(* CODESYS project basevista.library
   Company: Vistaprint
   Title: Base_PLC
   Description: 0.3.4.8 - Bug fix alarm entry,reset and clear
      0.3.4.7 - Increased the maxchildnumber to 40
      0.3.4.6 - Increased the maxchildnumber to 40
      0.3.4.5 - BugFix in alarm manager
      0.3.4.2 - Changed the Pramas Text in FB_CtrlBase
      0.3.4.1 - State single answer. Reset pending alarm class to NONE.
      0.3.4.0 - New CheckAllChildState also true feedback if check state of child OFF or EOFF and child in ERROR;
      - Bug fix Always Single-answer and startup with wait on PON
      - FB_Alm_Man: New Property IsInitDone		feedback at least one valid time stamp read out 
      0.3.3.7 - CheckParentAlmClass OFF and STOP added -> reaction of Controller
      0.3.3.6 - FB_Alm_Man Property CntPerClass added, alarm classes EOFF, OFF and STOP from parent to child, in EOFFBusy and OFF busy command in cyclic action (not entry action)
      
      0.3.3.4 - Added IO support for USINT datatype
      
      0.3.3.3 - Bug fixed in getInBolDebounced(FUN)
      
      0.3.3.2 - New function setAllCtrlAlarmFB -> all controller init pointer of alarmhandler; 
      - Rename GetInUint ->getInUint; 
      - New function ScaleINT (scale integer variable p.e. analog increment to 0.1mm)
      
      0.3.3.1  Added getInBolDebounced(FUN) and T_Ctrl_IoBoolDebounced(STRUCT) for debouncing inputs
      0.3.3.0 - Added pfbAlarmCtrl and the "zugehörige" property to allow clean alarm calls also from controllers in libraries.
      0.3.2.0 - Del getCtrlCIF,iniCtrlArray; Set cmds to child EOFF,OFF,PON; EOFF State; Check child ALM EOFF     
      0.3.1.3 - Bugfix
      0.3.1.2 - Added iniAllCtrlArrays - this is iniCtrlArray + the cif array
      0.3.1 - Added the automatic EOff propagation.
      0.3.0 - Added the substate to T_CTRL_CLASS_STATEMACHINE
      Automatic Substate handling.
      0.2.3 - Added support for sub usec cycletimes
      0.2.2 - Added the UInt for IO. T_CTRL_IOUint, setInUint(), setOutUint()
      0.2.1 - Added the property CtrlCIf to FB_CtrlBase
   Version: 0.3.4.8

Project tree, tasks and I/O mapping:
  libraries: Tc2_Standard, 3.3.0.0 (Beckhoff Automation GmbH); Tc2_System, 3.3.5.0 (Beckhoff Automation GmbH); Tc2_Utilities, 3.3.7.0 (Beckhoff Automation GmbH); Tc3_Interfaces, 3.3.0.0 (Beckhoff Automation GmbH); Tc3_MemMan, 3.3.1.0 (Beckhoff Automation GmbH); Tc3_Module, 3.3.5.0 (Beckhoff Automation GmbH)
  POUs/
    Alarm/
      data type E_AlmClass
      data type E_AlmCmd
      data type E_AlmState
      function block FB_Alm_Man [ST]: aCntPerClass, clearAlarm, IsInitDone, setAlarm
      data type T_AlmElement
      data type T_Ctrl_Alm
    BaseCtrl/
      global variables Base_CmdState
      global variables Base_Const
      data type E_Mode
      function block FB_CtrlBase [ST]: AddChild, AlarmCtrl, Always, CheckAllChildAlmClass, CheckAllChildState, CheckChildAlmClass, CheckCmdValid, CheckParentAlmClass, CtrlCIf, CtrlFB, CtrlInit, CycleEndDuty, CycleStartDuty, EOFF_EntryAction, FB_init, getCmdState, iniAllCtrlArrays, IoInBridge, IoOutBridge, SetAllChildAlmClass, SetAllChildCmd, sta_EOFF, sta_EOFFBusy, sta_ERROR, sta_ERRORQuit, sta_OFF, sta_OFFBusy, sta_PON, sta_PONBusy, sta_SINGLE_ANSWER, StateMachine
      interface I_CtrlBase: CtrlCIf, CtrlFB
      data type T_Ctrl_CIf
      data type T_Ctrl_Class
      data type T_Ctrl_Class_Alm
      data type T_Ctrl_Class_StateMachine
      data type T_Ctrl_CmdListElement
      data type T_Ctrl_Info
      data type T_Ctrl_IoBool
      data type T_Ctrl_IoBoolDebounced
      data type T_Ctrl_IoInt
      data type T_Ctrl_IoUint
      data type T_Ctrl_IoUsint
      data type T_Ctrl_Job
      data type T_Ctrl_SwCfg
      data type T_fbInfo
    Utility/
      DLL (Double Linked List)/
        function block FB_DLL [ST]: addElement, deleteAll, deleteElement, FB_init, firstElement, numberOfElements, searchElement
        data type T_Element
      function getInBol [ST]
      function getInBolDebounced [ST]
      function getInInt [ST]
      function getInUint [ST]
      function getInUsint [ST]
      function getStrInstanceName [ST]
      function ScaleINT [ST]
      function setAllCtrlAlarmFB [ST]
      function setOutBol [ST]
      function setOutInt [ST]
      function setOutUint [ST]
      function setOutUsint [ST]
  Version/
    global variables Global_Version
*)

// POUs/Alarm/E_AlmClass
TYPE E_AlmClass :
(
	///no alarm active
	NONE := 0,
	///info
	INFO,
	///warning
	WARNING,
	///tact stop
	TSTOP,
	///stop
	STOP,
	///off
	OFF,
	///Emergency off
	EOFF,
	Max_E_AlmClass
) INT;
END_TYPE

// POUs/Alarm/E_AlmCmd
TYPE E_AlmCmd :
(
	DONE := -1,
	INITIALIZED := 0,
	RESET_ALL := 2,
	RESET_RST := 4,
	RESET_CLR := 6,
	Max_E_AlmCmd
);
END_TYPE

// POUs/Alarm/E_AlmState
TYPE E_AlmState :
(
	///no alarm active
	NONE := 0,
	///alarm clear entry -> set bit1
	CLR := 1,
	///entry resettable alarm ->  set bit2
	RST := 2,
	///entry non resettable alarm ->  set bit2 + bit3
	SET := 3,
	Max_E_AlmState
);
END_TYPE

// POUs/Alarm/T_AlmElement
TYPE T_AlmElement :
STRUCT
	///unique alarm number := 100000*udiMachineNr + intCtrlId*100 + udiAlarmNr
	udiNr: UDINT;
	///additional information - better string???
	dinInfo: DINT;
	///corresponding alarm class
	eClass: E_AlmClass;
	///clear, resetable
	intState: E_AlmState;
	///entry time
	strDTEntry: STRING;
	///from machine (standard = 1)
	udiMachineNr: UDINT;
	///from controller
	intCtrlId: INT;
	///local alarm number
	udiAlarmNr: UDINT;
	// for debugging string alarm controller-alarm
	strText: STRING;
END_STRUCT
END_TYPE

// POUs/Alarm/T_Ctrl_Alm
TYPE T_Ctrl_Alm :
STRUCT
	///alarm flag array
	bol: BOOL;
	eAlmClass: E_AlmClass;
	strText: STRING;
END_STRUCT
END_TYPE

// POUs/BaseCtrl/E_Mode
{attribute 'qualified_only' := ''}
TYPE E_Mode :
(
	INITIALIZED := 0,
	AUTO := 10,
	SEMI := 11,
	MANU := 12
) INT;
END_TYPE

// POUs/BaseCtrl/T_Ctrl_CIf
TYPE T_Ctrl_CIf :
STRUCT
	Job: T_Ctrl_Job;
	Info: T_Ctrl_Info;
	SwCfg: T_Ctrl_SwCfg;
END_STRUCT
END_TYPE

// POUs/BaseCtrl/T_Ctrl_Class
TYPE T_Ctrl_Class :
STRUCT
	///local test flag to supress cyclic run (for debugging after init)
	bolActivate					: BOOL;
	intCmd						: INT;
	intCmdLast					: INT;
	eModeHistory				: E_Mode;
	///local flag mode change detected
	bolChangeBackToAUTO			: BOOL;
	StateMachine				: T_Ctrl_Class_StateMachine;
	SubStateMachine				: T_Ctrl_Class_StateMachine;
	Alarm						: T_Ctrl_Class_Alm;
	FUBInfo						: T_fbInfo;
END_STRUCT
END_TYPE

// POUs/BaseCtrl/T_Ctrl_Class_Alm
TYPE T_Ctrl_Class_Alm :
STRUCT
	bolResetOk: BOOL;
	///flag positive check me alarm from child
	bolfp: BOOL;
	///local activ alarm class of parent ctrl
	eParent_ActivAlmClass: E_AlmClass;
	///highest local activ alarm class
	eActivAlmClass: E_AlmClass;
END_STRUCT
END_TYPE

// POUs/BaseCtrl/T_Ctrl_Class_StateMachine
TYPE T_Ctrl_Class_StateMachine :
STRUCT
	///actual state
	intState: INT;
	///state of last cycle
	intStateLastCycle: INT;
	///save history backup p.e. in ERROR state
	intStateHistory: INT;
	///set state for next cycle
	intStateNext: INT;
	///[ms] to simulate state in SINGLE_ANSWER
	udiStateSimSetTime_ms: UDINT := 1000;
	///[ms] time in one state
	udiTimeInState_ms: UDINT;
	///[ms] time in one state
	relTimeInState_ms: REAL;
	///[us] time in one state
	udiTimeInState_us: UDINT;
END_STRUCT
END_TYPE

// POUs/BaseCtrl/T_Ctrl_CmdListElement
TYPE T_Ctrl_CmdListElement :
STRUCT
	///command implemented in controller
	intCmd: INT;
	///command is available info for UI
	bolAvailable: BOOL;
	/// Name of command. Important for UI.
	strName: STRING(80);
END_STRUCT
END_TYPE

// POUs/BaseCtrl/T_Ctrl_Info
TYPE T_Ctrl_Info :
STRUCT
	///name of controller instance
	strName				: STRING(80);
	///class of controller
	strType				: STRING(80);
	///unique controller instance identification number
	intCtrlId			: INT;
	///unique identification number of parent controller instance
	intParentCtrlId		: INT;
	///all inputs valid -> init done
	bolInitDone			: BOOL;
	///Childs
	p_afbChild			: ARRAY[0..Base_Const.cMaxNrOfChilds] OF POINTER TO FB_CtrlBase;
	///common interface array of childs
	p_aCIf				: ARRAY[0..Base_Const.cMaxNrOfChilds] OF POINTER TO T_Ctrl_CIf;
	/// Child Count
	uinChildNbr			: UINT;
END_STRUCT
END_TYPE

// POUs/BaseCtrl/T_Ctrl_IoBool
TYPE T_Ctrl_IoBool :
STRUCT
	///mapped io variable to hardware
	map: BOOL;
	///shows the state of (input: mapped, output: set by programm respectiv at the moment one cycle later evtl. from the forcing if forcing active) -> necessary for what?
	state: BOOL;
	///variabel to/ from program
	intern: BOOL;
	///variabel set from UI
	force: BOOL;
	///enable force of single io-datapoint
	EnForce: BOOL;
END_STRUCT
END_TYPE

// POUs/BaseCtrl/T_Ctrl_IoBoolDebounced
TYPE T_Ctrl_IoBoolDebounced :
STRUCT
	///mapped io variable to hardware
	map: BOOL;
	///shows the state of (input: mapped, output: set by programm respectiv at the moment one cycle later evtl. from the forcing if forcing active) -> necessary for what?
	state: BOOL;
	///variabel to/ from program
	intern: BOOL;
	///variabel set from UI
	force: BOOL;
	///enable force of single io-datapoint
	EnForce: BOOL;
	// time since last input change
	udinDebouncedTimeCounter_ms: UDINT;
END_STRUCT
END_TYPE

// POUs/BaseCtrl/T_Ctrl_IoInt
TYPE T_Ctrl_IoInt :
STRUCT
	///mapped io variable to hardware
	map: INT;
	///shows the state of (input: mapped, output: set by programm respectiv at the moment one cycle later evtl. from the forcing if forcing active) -> necessary for what?
	state: INT;
	///variabel to/ from program
	intern: INT;
	///variabel set from UI
	force: INT;
	///enable force of single io-datapoint
	EnForce: BOOL;
END_STRUCT
END_TYPE

// POUs/BaseCtrl/T_Ctrl_IoUint
TYPE T_Ctrl_IoUint :
STRUCT
	///mapped io variable to hardware
	map: UINT;
	///shows the state of (input: mapped, output: set by programm respectiv at the moment one cycle later evtl. from the forcing if forcing active) -> necessary for what?
	state: UINT;
	///variabel to/ from program
	intern: UINT;
	///variabel set from UI
	force: UINT;
	///enable force of single io-datapoint
	EnForce: BOOL;
END_STRUCT
END_TYPE

// POUs/BaseCtrl/T_Ctrl_IoUsint
TYPE T_Ctrl_IoUsint :
STRUCT
	///mapped io variable to hardware
	map: USINT;
	///shows the state of (input: mapped, output: set by programm respectiv at the moment one cycle later evtl. from the forcing if forcing active) -> necessary for what?
	state: USINT;
	///variabel to/ from program
	intern: USINT;
	///variabel set from UI
	force: USINT;
	///enable force of single io-datapoint
	EnForce: BOOL;
END_STRUCT
END_TYPE

// POUs/BaseCtrl/T_Ctrl_Job
TYPE T_Ctrl_Job :
STRUCT
	///mode if mode = AUTO -> ACmd will be used, otherwise the MCmd channel is open
	eMode: E_Mode;
	///automatic command from parent ctrl
	intACmd: INT;
	///manual command from UI p.e.
	intMCmd: INT;
	///active cmd
	strCmd: STRING;
	///active state
	intState: INT;
	strState: STRING;
	///if used - show substates for debugging
	strSubState: STRING;
	///event channel to signal special events to parent parallel to status
	intEvt: INT;
	///reset all alarms
	bolAlmReset: BOOL;
	///activate io-forcing
	bolIoForce: BOOL;
	///overwrite suspend all interlocks (for debugging/testing)
	bolIlkOverwrite: BOOL;
	///activ alarm class of parent ctrl
	eParent_ActivAlmClass: E_AlmClass;
	///activ alarm class of me ctrl
	eMe_ActivAlmClass: E_AlmClass;
	///list of all implemented commands
	aCmdList: ARRAY[0..cMaxCmdPerCtrl] OF T_Ctrl_CmdListElement;
END_STRUCT
END_TYPE

// POUs/BaseCtrl/T_Ctrl_SwCfg
TYPE T_Ctrl_SwCfg :
	STRUCT
		///hardware/controller exists
		bolExist: BOOL;
		///enable statemachine
		bolEnable: BOOL;
		///set controller in simulation(statemachine active, io local simulated)
		bolSimulation: BOOL;
	END_STRUCT
END_TYPE

// POUs/BaseCtrl/T_fbInfo
TYPE T_fbInfo :
STRUCT
	bolCycleTimeBelowMS			: BOOL;
	udiSample_ms				: UDINT;
	udiSample_us				: UDINT;
END_STRUCT
END_TYPE

// POUs/Utility/DLL (Double Linked List)/T_Element
{attribute 'enable_dynamic_creation' := ''}
TYPE T_Element :
STRUCT
	pPrevElement: POINTER TO T_Element;
	pData: POINTER TO BYTE;
	uliKey: ULINT;
	pNextElement: POINTER TO T_Element;
END_STRUCT
END_TYPE

// POUs/BaseCtrl/Base_CmdState
VAR_GLOBAL CONSTANT
	///ctrl commands definitions
	///general commands 2-200 - every command has to be a even number
	cCMD_DONE: INT := -1;
	cCMD_INITIALIZED: INT := 0;
	cCMD_PON: INT := 2;
	cCMD_EOFF: INT := 4;
	cCMD_OFF: INT := 6;
	cCMD_INIT: INT := 8;
	cCMD_RUN: INT := 10;
	cCMD_STOP: INT := 12;
	cCMD_TSTOP: INT := 14;
	///ctrl states definitions
	cSTA_DONE: INT := cCMD_DONE;
	cSTA_INITIALIZED: INT := cCMD_INITIALIZED;
	cSTA_PONBusy: INT := 1;
	cSTA_PON: INT := cCMD_PON;
	cSTA_EOFFBusy: INT := 3;
	cSTA_EOFF: INT := cCMD_EOFF;
	cSTA_OFFBusy: INT := 5;
	cSTA_OFF: INT := cCMD_OFF;
	cSTA_INITBusy: INT := 7;
	cSTA_INIT: INT := cCMD_INIT;
	cSTA_RUNBusy: INT := 9;
	cSTA_RUN: INT := cCMD_RUN;
	cSTA_STOPBusy: INT := 11;
	cSTA_STOP: INT := cCMD_STOP;
	cSTA_TSTOPBusy: INT := 13;
	cSTA_TSTOP: INT := cCMD_TSTOP;
	///special states without corresponding cmd
	cSTA_ERROR: INT := 150;
	cSTA_ERRORQuit: INT := 151;
	cSTA_SINGLE_ANSWER: INT := 152;
END_VAR

// POUs/BaseCtrl/Base_Const
VAR_GLOBAL CONSTANT
	///number of child access possible in one controller class
	cMaxNrOfChilds: UINT := 25;
	///maximal number of commands implemented in one controller class
	cMaxCmdPerCtrl: UINT := 15;
	///maximal number of commands implemented in one controller class
	cMaxBaseCmdState: UINT := 200;
END_VAR

// Version/Global_Version
// This function has been automatically generated from the project information.
VAR_GLOBAL CONSTANT
	{attribute 'const_non_replaced'}
	stLibVersion_Base_PLC : ST_LibVersion := (iMajor := 0, iMinor := 3, iBuild := 4, iRevision := 8, sVersion := '0.3.4.8');
END_VAR

// POUs/Alarm/FB_Alm_Man
FUNCTION_BLOCK FB_Alm_Man
VAR_INPUT
	;
END_VAR
VAR_IN_OUT
	bolCtrlRst: BOOL; // reset all controller
END_VAR

VAR CONSTANT
	/// config alarm handler number of elements of queue
	c_uinMaxAlmElements: UINT := 99;
	/// 0: with history on PLC, auto clr alarms from array if alarm state clear is set
	c_uinModeAlarm: UINT := 1;
	/// machine number 1, at the moment every time set to 1
	c_udiMachineNr: UDINT := 1;
	/// commands from the UI
	cCMD_RESET_ALL: INT := 2;
	/// reset state=RST, reset state CLR
	cCMD_RESET_RST: INT := 4;
	/// reset state CLR -> c_uinModeAlarm = 1, automatic reset will be done on PLC
	cCMD_RESET_CLR: INT := 6;
END_VAR
VAR
	///------------------------------------------------------------
	/// UI interface
	/// alarmarray PLC -> UI
	aAlm: ARRAY[0..c_uinMaxAlmElements] OF T_AlmElement;
	/// command interface for UI -> PLC
	intAlmCmd: INT;
	///------------------------------------------------------------
	/// real local variables
	fbGetLocalTime: NT_GetTime;
	strActTime: STRING;
	jj: UINT;
	EmptyAlmElement: T_AlmElement;
	intState: INT;
	intTestCtrl: INT := 12;
	intTestState: INT;
	udiTestAlarmNr: UDINT;
	dinTestInfo: DINT;
	aCtrlAlm: ARRAY[1..6] OF T_Ctrl_Alm;
	eActiveAlmClass: E_AlmClass;

	aCntActiveAlmPerClass: ARRAY[0..(E_AlmClass.Max_E_AlmClass-1)] OF UINT; // count off all active alarms per class, idx=0 all active alarms
	bolTimeReadDone : BOOL;
	bolTimeStampValid : BOOL;
END_VAR

(*__________________________________________________________________________________________________
¦	
¦	Vistaprint Schweiz GmbH
¦	CH - 8401 Winterthur
¦
¦	www.vistaprint.ch - info@vistaprint.ch
¦___________________________________________________________________________________________________

Function desription:
The alarm manager sets and clears alarms from the internal array. In the internal array all active 
alarms of a machine are listed. The list has no order. A new entry will be inserted at the next 
free place.

For the easy usage for UI the function block is to be define as global. And then the cmd for reset should be 
set when the button is pressed -> intAlmCmd = cCMD_RESET_ALL
All active alarms are shown in the aAlm array.

History:
Version		Date			Author		Comment
---------------------------------------------------------------------------------------------------
0.00.1		29.04.2013		AVME/KVO	Start history
0.00.2		06.01.2014		AVME/PRE	Implement the counted active messages array
0.00.3		17.02.2014		AVME/KVO	New Property IsInitDone 
										feedback at least one valid time stamp read out 
										-> check at startup before cyclic call of FB's to avoid alarms without valid timestamp
0.00.4		16.05.2014		AVME/DSC	-> Inserted new "setAlarm" Method from Patrik C. (code review)									
										-> BugFix, build sum of all active alarms
___________________________________________________________________________________________________*)

// read out actual TIME
fbGetLocalTime.NETID := '';
fbGetLocalTime.START := NOT bolTimeReadDone;
fbGetLocalTime.TMOUT := T#5S;
fbGetLocalTime();

IF (fbGetLocalTime.START=TRUE) THEN
	IF  ((fbGetLocalTime.Busy=FALSE) AND (fbGetLocalTime.ERR=FALSE)) THEN
		bolTimeReadDone := TRUE;
		strActTime := TC2_UTILITIES.SYSTEMTIME_TO_STRING(fbGetLocalTime.TIMESTR); // YYYY-MM-DD-hh:mm:ss.xxx
		bolTimeStampValid := TRUE; // -> entry alarms with valid time stamp
	END_IF
ELSE
	bolTimeReadDone := FALSE;
END_IF


// interface for UI access
CASE intState OF
	
	0: // reset cmd
		intAlmCmd := cCMD_DONE; // Ready for new cmd
		intState := intState + 1;
		
	1: // wait for cmd
		IF (intAlmCmd=cCMD_RESET_ALL) OR (intAlmCmd=cCMD_RESET_CLR) OR  (intAlmCmd=cCMD_RESET_RST) THEN
			intState := intState + 1;
		END_IF
		
	2: // reset alarms
		// reset state=RST, reset state CLR
		THIS^.clearAlarm(((intAlmCmd=cCMD_RESET_ALL) OR (intAlmCmd=cCMD_RESET_RST)), TRUE);
		intState := intState + 1;
		
	3: // reset state machines
		bolCtrlRst := TRUE;
		intState := 0; // done

END_CASE

// build sum of all active alarms
aCntActiveAlmPerClass[0] := 0;
FOR jj:= 1 TO INT_TO_UINT(E_AlmClass.Max_E_AlmClass-1) BY 1 DO
	aCntActiveAlmPerClass[0] := aCntActiveAlmPerClass[0] + aCntActiveAlmPerClass[jj];
END_FOR

//**********************************************************************************************
// Test manual set/reset/clear alarm
//**********************************************************************************************
CASE intTestState OF
	
	0: // wait
		
	1: //CLR
		THIS^.setAlarm(intTestCtrl,udiTestAlarmNr,dinTestInfo,ADR(aCtrlAlm),E_AlmState.CLR,eActiveAlmClass);
		intTestState := 0;
		
	2: // RST
		THIS^.setAlarm(intTestCtrl,udiTestAlarmNr,dinTestInfo,ADR(aCtrlAlm),E_AlmState.RST,eActiveAlmClass);
		intTestState := 0;
		
	3: // SET
		THIS^.setAlarm(intTestCtrl,udiTestAlarmNr,dinTestInfo,ADR(aCtrlAlm),E_AlmState.SET,eActiveAlmClass);
		intTestState := 0;

END_CASE

PROPERTY PUBLIC aCntPerClass : ARRAY[0..(E_AlmClass.Max_E_AlmClass-1)] OF UINT
GET
aCntPerClass := aCntActiveAlmPerClass;
END_GET
END_PROPERTY

METHOD clearAlarm : BOOL
VAR_INPUT
	///-> clear all entries with state RST
	bolClear_RST: BOOL;
	///-> clear all entries with state CLR
	bolClear_CLR: BOOL;
END_VAR
VAR
	ii: UINT;
END_VAR
FOR ii:= 0 TO INT_TO_UINT(E_AlmClass.Max_E_AlmClass-1) BY 1 DO
	aCntActiveAlmPerClass[ii] := 0; // reset alarm counter
END_FOR

FOR ii:= 0 TO c_uinMaxAlmElements BY 1 DO
	
	IF (aAlm[ii].udiNr>0) THEN 
		
		IF (((aAlm[ii].intState=E_AlmState.RST) AND (bolClear_RST)) OR
			((aAlm[ii].intState=E_AlmState.CLR) AND (bolClear_CLR)))THEN
			
			aAlm[ii] := EmptyAlmElement; // clear entry
		ELSE
			//count alarms per class
			aCntActiveAlmPerClass[aAlm[ii].eClass] := aCntActiveAlmPerClass[aAlm[ii].eClass] + 1; 
		END_IF
		
	END_IF
END_FOR
END_METHOD

PROPERTY IsInitDone : BOOL
GET
// feedback at least one valid time stamp read out 
//-> check at startup before cyclic call of FB's to avoid alarms without valid timestamp
IsInitDone := bolTimeStampValid;
END_GET
END_PROPERTY

METHOD setAlarm : E_AlmClass
VAR_INPUT
	///from controller 
	intCtrlId: INT;
	///local alarm number
	udiAlarmNr: UDINT;
	///additional information - string???
	dinInfo: DINT;
	///corresponding alarm class
	p_Ctrl_Alm: POINTER TO T_Ctrl_Alm;
	///clear, resetable
	intState: E_AlmState;
END_VAR
VAR_IN_OUT
	eMe_ActivAlmClass: E_AlmClass;
END_VAR
VAR
	InAlmElement: T_AlmElement;
	ii: UINT;
	e_LocAlmClass: E_AlmClass;
END_VAR
// chack if pointer valid
IF (p_Ctrl_Alm <> Tc3_MemMan.NULL) AND (udiAlarmNr>0) THEN 
	e_LocAlmClass := p_Ctrl_Alm[udiAlarmNr-1].eAlmClass;
ELSE
	// novalid pointer reached!!
   	e_LocAlmClass := E_AlmClass.EOFF; 
END_IF
 
// Copy alarm input data to local alm struct
InAlmElement.udiMachineNr := c_udiMachineNr;
InAlmElement.intCtrlId := intCtrlId;
InAlmElement.udiAlarmNr := udiAlarmNr;
InAlmElement.udiNr := 100000*InAlmElement.udiMachineNr + INT_TO_UDINT(100*InAlmElement.intCtrlId) + InAlmElement.udiAlarmNr;
InAlmElement.dinInfo := dinInfo;
InAlmElement.eClass := e_LocAlmClass;
InAlmElement.intState := intState;
InAlmElement.strDTEntry := strActTime;
InAlmElement.strText := p_Ctrl_Alm[udiAlarmNr-1].strText;

ii := 0;
//KVO 7.7.2014 AND (aAlm[ii].udiNr <> 0) removed from while because there could be entries above a cleared alarm!
WHILE (ii <= c_uinMaxAlmElements)  AND (InAlmElement.udiNr <> aAlm[ii].udiNr) DO
	ii := ii + 1;              
END_WHILE
 
IF (ii <= c_uinMaxAlmElements) THEN
	
	// Alarm already exist
	IF (aAlm[ii].udiNr = InAlmElement.udiNr) THEN
		CASE InAlmElement.intState OF
			E_AlmState.SET, E_AlmState.RST:
				// refresh state, alarm additional info
				aAlm[ii].dinInfo := InAlmElement.dinInfo;
				aAlm[ii].intState := InAlmElement.intState;
			E_AlmState.CLR:
				IF (aCntActiveAlmPerClass[aAlm[ii].eClass]>0) THEN
					aCntActiveAlmPerClass[aAlm[ii].eClass] := aCntActiveAlmPerClass[aAlm[ii].eClass] - 1; 
				END_IF
				
				IF (c_uinModeAlarm=1) THEN // no history on PLC
					aAlm[ii] := EmptyAlmElement; // clear entry
				ELSE
					aAlm[ii].intState := E_AlmState.CLR; // set clear state -> entry in plc history if needed
				END_IF
		END_CASE          
	END_IF
	
	// New Alarm entry
	IF (aAlm[ii].udiNr = 0) THEN
		CASE InAlmElement.intState OF
			E_AlmState.SET, E_AlmState.RST:
				aAlm[ii] := InAlmElement;
				//count alarms per class
				aCntActiveAlmPerClass[aAlm[ii].eClass] := aCntActiveAlmPerClass[aAlm[ii].eClass] + 1; 
	
				IF (InAlmElement.eClass>eMe_ActivAlmClass) THEN 
					eMe_ActivAlmClass := InAlmElement.eClass;
				END_IF
		END_CASE
	END_IF
	
END_IF
END_METHOD

END_FUNCTION_BLOCK

// POUs/BaseCtrl/FB_CtrlBase
{attribute 'reflection'}
FUNCTION_BLOCK FB_CtrlBase IMPLEMENTS I_CtrlBase
VAR
	// common interface struct for public access
	CIf				: T_Ctrl_CIf;

	// pointer to global alarm handler function block 
	pfbAlarmCtrl	: POINTER TO FB_Alm_Man;
 
	// basic local controller class struct
	me	: T_Ctrl_Class;
	fbSimulationTimer	: TON;
	{attribute 'noinit'}
	{attribute 'instance-path'}
	strMyInstancePath: STRING;
END_VAR

(*__________________________________________________________________________________________________
¦	
¦	Vistaprint Schweiz GmbH
¦	CH - 8401 Winterthur
¦
¦	www.vistaprint.ch - info@vistaprint.ch
¦___________________________________________________________________________________________________

Function desription:
Basic controller implementation. This Controller should be the base father controller for all in the
feature implemented ctontroller classes.


History:
Version		Date			Author		Comment
---------------------------------------------------------------------------------------------------
0.00.1		25.04.2013		AVME/KVO	Start history
0.00.2		06.01.2014		AVME/PRE	Alarmclasses EOFF, OFF and STOP are send to parent and childs
0.00.3		08.01.2014		AVME/KVO	CheckParentAlmClass OFF and STOP added -> reaction of Controller
0.00.4		04.02.2014		AVME/KVO	New CheckAllChildState also true feedback if check state of 
										child OFF or EOFF and child in ERROR
0.00.5		17.02.2014		AVME/KVO	Bug fix Always Single-answer and startup with wait on PON before change 
										state to EOFFBusy and so on
										Bug fix in CheckParentAlmClass not reset command PON
0.00.6		26.02.2014		AVME/DSC	State single answer. Reset pending alarm class to NONE.

___________________________________________________________________________________________________*)


IF (me.bolActivate) THEN // cyclic call enabled
	
	IF (CIf.Info.bolInitDone=FALSE) THEN // first cycle -> init
		CtrlInit();
		CIf.Info.bolInitDone := TRUE;
	ELSE
		CycleStartDuty();
	
		Always();
		
		StateMachine();
		
		CycleEndDuty();
	END_IF
	
END_IF;

METHOD PROTECTED AddChild : POINTER TO T_Ctrl_CIf;
VAR_INPUT
	p_fbChild			: I_CtrlBase;
END_VAR
AddChild := 0;

IF CIf.Info.uinChildNbr <= Base_Const.cMaxNrOfChilds THEN
	CIf.Info.p_afbChild[CIf.Info.uinChildNbr] := p_fbChild.CtrlFB;
	CIf.Info.p_aCIf[CIf.Info.uinChildNbr] := CIf.Info.p_afbChild[CIf.Info.uinChildNbr]^.CtrlCIf;
	CIf.Info.p_aCIf[CIf.Info.uinChildNbr]^.Info.intParentCtrlId := CIf.Info.intCtrlId;
	CIf.Info.uinChildNbr := CIf.Info.uinChildNbr + 1;
	AddChild := p_fbChild.CtrlCIf;
END_IF
END_METHOD

PROPERTY PUBLIC AlarmCtrl : POINTER TO FB_Alm_Man
SET
pfbAlarmCtrl := AlarmCtrl;
END_SET
END_PROPERTY

METHOD PROTECTED Always : BOOL
// ----------------------------------------------------------------------------------
// cyclic actions outside of statemachine
IF (me.StateMachine.intState<>cSTA_SINGLE_ANSWER) THEN
	
	; // always error supervision
	// ---------------------------------------------------------------------------------
END_IF

// ----------------------------------------------------------------------------------
// Conditions Always
IF (me.bolChangeBackToAUTO=TRUE) THEN // switch mode to automatic switch off controller
	me.StateMachine.intStateNext := cSTA_OFFBusy;
	me.bolChangeBackToAUTO := FALSE;
END_IF

IF (CIf.SwCfg.bolExist=FALSE) THEN // hardware of controller does not exist
	me.StateMachine.intStateNext := cSTA_SINGLE_ANSWER;
ELSE
	IF (((me.StateMachine.intState=cSTA_INITIALIZED) OR (me.intCmd=cCMD_PON)) 
		AND (me.StateMachine.intState<>cSTA_PONBusy) AND (me.StateMachine.intState<>cSTA_PON)
		AND (me.StateMachine.intState<>cSTA_ERROR) AND (me.StateMachine.intState<>cSTA_ERRORQuit) 
		AND (me.StateMachine.intState<>cSTA_EOFF) AND (me.StateMachine.intState<>cSTA_EOFFBusy)) THEN // switch after startup to PONBusy
		me.StateMachine.intStateNext := cSTA_PONBusy;
		
	ELSIF (((me.Alarm.eActivAlmClass=E_AlmClass.EOFF) OR (me.intCmd=cCMD_EOFF)) 
		AND (me.StateMachine.intState<>cSTA_ERROR) AND (me.StateMachine.intState<>cSTA_ERRORQuit) 
		AND (me.StateMachine.intState<>cSTA_EOFF) AND (me.StateMachine.intState<>cSTA_EOFFBusy)
		AND (me.StateMachine.intState>cSTA_PON)) THEN
		me.StateMachine.intStateNext := cSTA_EOFFBusy;
	
	ELSIF (((me.Alarm.eActivAlmClass=E_AlmClass.OFF) OR (me.intCmd=cCMD_OFF))
		AND (me.StateMachine.intState<>cSTA_ERROR) AND (me.StateMachine.intState<>cSTA_ERRORQuit)
		AND (me.StateMachine.intState<>cSTA_EOFF) AND (me.StateMachine.intState<>cSTA_EOFFBusy)
		AND (me.StateMachine.intState<>cSTA_OFF) AND (me.StateMachine.intState<>cSTA_OFFBusy)
		AND (me.StateMachine.intState>cSTA_PON)) THEN
		me.StateMachine.intStateNext := cSTA_OFFBusy;
	
	END_IF
END_IF
END_METHOD

METHOD PROTECTED CheckAllChildAlmClass : BOOL
VAR_INPUT
	In_intCheckAlmClass : INT;
END_VAR
VAR
	uinIdx: UINT;
END_VAR
// check if at least one child has actual this alarm class active
CheckAllChildAlmClass := FALSE;

IF (CIf.Info.uinChildNbr > 0) THEN
	FOR uinIdx := 0 TO CIf.Info.uinChildNbr - 1 DO
		CheckAllChildAlmClass := (CIf.Info.p_aCIf[uinIdx]^.Job.eMe_ActivAlmClass = In_intCheckAlmClass);
		IF (CheckAllChildAlmClass=TRUE) THEN // at least one child has actual this alarm class active
			EXIT;
		END_IF
	END_FOR
END_IF
END_METHOD

METHOD PROTECTED CheckAllChildState : BOOL;
VAR_INPUT
	In_intCheckState : INT;
END_VAR
VAR
	uinIdx: UINT;
END_VAR
// check if all child controller have reached the final In_intCheckState
CheckAllChildState := TRUE;
IF (CIf.Info.uinChildNbr > 0) THEN
	FOR uinIdx := 0 TO CIf.Info.uinChildNbr - 1 DO
		IF ((In_intCheckState<>cSTA_EOFF) AND (In_intCheckState<>cSTA_OFF)) THEN
			CheckAllChildState := CheckAllChildState AND (CIf.Info.p_aCIf[uinIdx]^.Job.intState = In_intCheckState);
		ELSE
			// if controlled state is OFF or EOFF and child is in ERROR -> answer state reached
			CheckAllChildState := (CheckAllChildState AND ((CIf.Info.p_aCIf[uinIdx]^.Job.intState = In_intCheckState) OR (CIf.Info.p_aCIf[uinIdx]^.Job.intState = cSTA_ERROR)));
		END_IF
		IF (CheckAllChildState=FALSE) THEN	// at least one child has not whished state reached
			EXIT ;
		END_IF 
	END_FOR
END_IF
END_METHOD

METHOD CheckChildAlmClass : BOOL
VAR_INPUT
;
END_VAR
VAR
;
END_VAR
//------------------------------------------------------------------------------------------------------
// check child alarm classes
// set me alarm class active if at least one child has an EOFF
IF CheckAllChildAlmClass(E_AlmClass.EOFF) THEN
	CIf.Job.eMe_ActivAlmClass := E_AlmClass.EOFF;
	me.Alarm.bolfp := TRUE;
ELSIF CheckAllChildAlmClass(E_AlmClass.OFF) THEN
	CIf.Job.eMe_ActivAlmClass := E_AlmClass.OFF;
	me.Alarm.bolfp := TRUE;
ELSIF CheckAllChildAlmClass(E_AlmClass.STOP) THEN
	CIf.Job.eMe_ActivAlmClass := E_AlmClass.STOP;
	me.Alarm.bolfp := TRUE;	
ELSE
	IF (me.Alarm.bolfp) THEN
		CIf.Job.eMe_ActivAlmClass := E_AlmClass.NONE; // no reset necessary
		me.Alarm.bolfp := FALSE;
	END_IF
END_IF

//------------------------------------------------------------------------------------------------------
// set alarm class parent of childs in the case of a parent or me=OFF or EOFF or STOP
IF (CIf.Job.eParent_ActivAlmClass=E_AlmClass.EOFF) OR (CIf.Job.eParent_ActivAlmClass=E_AlmClass.OFF) OR (CIf.Job.eParent_ActivAlmClass=E_AlmClass.STOP) THEN
	SetAllChildAlmClass(CIf.Job.eParent_ActivAlmClass);
ELSIF(CIf.Job.eMe_ActivAlmClass=E_AlmClass.EOFF) OR (CIf.Job.eMe_ActivAlmClass=E_AlmClass.OFF) OR (CIf.Job.eMe_ActivAlmClass=E_AlmClass.STOP) THEN
	SetAllChildAlmClass(CIf.Job.eMe_ActivAlmClass);
ELSE
	// no important alarm for child active
	SetAllChildAlmClass(E_AlmClass.NONE);
END_IF
END_METHOD

METHOD PRIVATE CheckCmdValid : BOOL
VAR
	ii: UINT;
END_VAR
CheckCmdValid := FALSE;
FOR ii:=0 TO cMaxCmdPerCtrl BY 1 DO
	// check if a valid cmd
	IF (CIf.Job.aCmdList[ii].intCmd=cCMD_INITIALIZED) OR (CIf.Job.aCmdList[ii].intCmd=cCMD_DONE) THEN
		EXIT; // end for
	END_IF
	// check if a in this ctrl implemented cmd
	IF (CIf.Job.aCmdList[ii].intCmd=me.intCmd) THEN
		CheckCmdValid := TRUE;
	END_IF
END_FOR
END_METHOD

METHOD PROTECTED CheckParentAlmClass : BOOL
// --------------------------------------------------------------------------
// check alarm recation class of master													
// --------------------------------------------------------------------------
IF (CIf.Job.eParent_ActivAlmClass = E_AlmClass.EOFF) THEN
	me.Alarm.eParent_ActivAlmClass := E_AlmClass.EOFF;
	// prevent automatic restart in manual or automatic
	IF (CIf.job.intACmd<>cCMD_PON) THEN // wait on startup until power on is ok
		CIf.job.intACmd := cCMD_DONE;
	END_IF
	
	IF (CIf.job.intMCmd<>cCMD_PON) THEN // wait on startup until power on is ok
		CIf.job.intMCmd := cCMD_DONE;
	END_IF
ELSIF (CIf.Job.eParent_ActivAlmClass = E_AlmClass.OFF) THEN
	me.Alarm.eParent_ActivAlmClass := E_AlmClass.OFF;
ELSIF (CIf.Job.eParent_ActivAlmClass = E_AlmClass.STOP) THEN
	me.Alarm.eParent_ActivAlmClass := E_AlmClass.STOP;
ELSE
	me.Alarm.eParent_ActivAlmClass := E_AlmClass.NONE;
END_IF
END_METHOD

PROPERTY PUBLIC CtrlCIf : POINTER TO T_Ctrl_CIf
GET
CtrlCIf := ADR(CIf);
END_GET
END_PROPERTY

PROPERTY PUBLIC CtrlFB : POINTER TO FB_CtrlBASE
GET
CtrlFB := ADR(THIS^);
END_GET
END_PROPERTY

METHOD PROTECTED CtrlInit : BOOL
VAR
	udiTaskCnt: UDINT;
	fbGETCURTASKINDEX: Tc2_System.GETCURTASKINDEX;
END_VAR

//automatic read out infos about FUB
udiTaskCnt := TwinCAT_SystemInfoVarList._AppInfo.TaskCnt;
fbGETCURTASKINDEX();
udiTaskCnt := fbGETCURTASKINDEX.index;
me.FUBInfo.udiSample_us := TwinCAT_SystemInfoVarList._TaskInfo[UDINT_TO_DINT(udiTaskCnt)].CycleTime/10; //[ms] X[100ns]/10 -> [us]
me.FUBInfo.udiSample_ms := TwinCAT_SystemInfoVarList._TaskInfo[UDINT_TO_DINT(udiTaskCnt)].CycleTime/10000; //[ms] X[100ns]/10000 -> [ms]
me.FUBInfo.bolCycleTimeBelowMS := me.FUBInfo.udiSample_us <= 1000;
END_METHOD

METHOD PROTECTED CycleEndDuty : BOOL

me.eModeHistory := CIf.Job.eMode;				// save mode to detect mode switches
me.intCmdLast := me.intCmd;
IF (me.StateMachine.intState<>cSTA_SINGLE_ANSWER) THEN // only if no simulation is active
	CIf.Job.intState := me.StateMachine.intState;		// set information of actual state to controller interface
	CIf.Job.strState := THIS^.getCmdState(intCmdState:=CIf.Job.intState,bolState:=TRUE);
ELSE
	CIf.Job.strState :=  TC2_STANDARD.CONCAT(STR1:='SINGLE_ANSWER-',STR2:=THIS^.getCmdState(intCmdState:=CIf.Job.intState,bolState:=TRUE));
END_IF

	
IF (me.StateMachine.intState<>me.StateMachine.intStateNext) THEN
	me.StateMachine.intState := me.StateMachine.intStateNext;  // set next state for next cycle
	me.StateMachine.udiTimeInState_ms := 0; // reset timer
	me.StateMachine.udiTimeInState_us := 0; // reset timer
	me.SubStateMachine.udiTimeInState_ms := 0; // reset timer
	me.SubStateMachine.udiTimeInState_us := 0; // reset timer
	me.SubStateMachine.intState := cSTA_DONE;
	// log state change -> open point
ELSE
	// increment time in state	
	me.StateMachine.udiTimeInState_us := me.StateMachine.udiTimeInState_us + me.FUBInfo.udiSample_us;
	me.StateMachine.udiTimeInState_ms := me.StateMachine.udiTimeInState_ms + me.FUBInfo.udiSample_ms;
	me.StateMachine.relTimeInState_ms := UDINT_TO_REAL(me.StateMachine.udiTimeInState_us) / 1000.0;
END_IF


IF (me.SubStateMachine.intState<>me.SubStateMachine.intStateNext) THEN
	me.SubStateMachine.intState := me.SubStateMachine.intStateNext;  // set next state for next cycle
	CIf.Job.strSubState := THIS^.getCmdState(intCmdState:=me.SubStateMachine.intState,bolState:=TRUE);
	me.SubStateMachine.udiTimeInState_ms := 0; // reset timer
	me.SubStateMachine.udiTimeInState_us := 0; // reset timer
	// log state change -> open point
ELSE
	// increment time in state	
	me.SubStateMachine.udiTimeInState_us := me.SubStateMachine.udiTimeInState_us + me.FUBInfo.udiSample_us;
	me.SubStateMachine.udiTimeInState_ms := me.SubStateMachine.udiTimeInState_ms + me.FUBInfo.udiSample_ms;
	me.SubStateMachine.relTimeInState_ms := UDINT_TO_REAL(me.SubStateMachine.udiTimeInState_us) / 1000.0;
END_IF
		
// --------------------------------------------------------------------------
// Final state reached -> reset command
// --------------------------------------------------------------------------
IF (CIf.Job.intState=me.intCmd) THEN 
	CIf.Job.intACmd := cCMD_DONE;
	CIf.Job.intMCmd := cCMD_DONE;
END_IF

// --------------------------------------------------------------------------
// reset local alarm class
// --------------------------------------------------------------------------
IF (CIf.Job.bolAlmReset=TRUE) AND (CIf.Job.intState<>cSTA_ERROR) AND (CIf.Job.intState<>cSTA_ERRORQuit) THEN
	CIf.Job.eMe_ActivAlmClass := E_AlmClass.NONE;
	CIf.Job.bolAlmReset := FALSE;
END_IF

// --------------------------------------------------------------------------
// output bridge
// --------------------------------------------------------------------------
THIS^.IoOutBridge();	// digitale and analoge outputs or forcing write to hardware
END_METHOD

METHOD PROTECTED CycleStartDuty : BOOL

	// --------------------------------------------------------------------------
	// input bridge
	// --------------------------------------------------------------------------
	THIS^.IoInBridge(); // digitale and analoge inputs read from hardware or forcing

	// --------------------------------------------------------------------------
	// check alarm recation class of master													
	// --------------------------------------------------------------------------
	THIS^.CheckParentAlmClass();
	
	// ----------------------------------------------------------------------------------
	// check the highest active alarm -> set local class
	// ----------------------------------------------------------------------------------
	IF (me.Alarm.eParent_ActivAlmClass>CIf.job.eMe_ActivAlmClass) THEN
		me.Alarm.eActivAlmClass := me.Alarm.eParent_ActivAlmClass;
	ELSE
		me.Alarm.eActivAlmClass := CIf.job.eMe_ActivAlmClass;
	END_IF
	
	// ----------------------------------------------------------------------------------
	// check child me and set parent alarm class
	// ----------------------------------------------------------------------------------
	CheckChildAlmClass();
	
	// --------------------------------------------------------------------------
	// get command											
	// --------------------------------------------------------------------------
	IF (CIf.Job.eMode = E_Mode.MANU) THEN
		me.intCmd := CIf.Job.intMCmd;  
	ELSE
		IF (me.eModeHistory <> E_MODE.AUTO) THEN
			CIf.Job.intMCmd:= cCMD_DONE;	// reset manual command
			me.bolChangeBackToAUTO := TRUE;	// switch off  or .....
		END_IF
		CIf.Job.eMode := E_MODE.AUTO;
		me.intCmd := CIf.Job.intACmd;
	END_IF
	CIf.Job.strCmd := THIS^.getCmdState(intCmdState:=me.intCmd,bolState:=FALSE);
END_METHOD

METHOD PROTECTED EOFF_EntryAction : BOOL
VAR_INPUT
END_VAR
 // used for special events in EOFF
END_METHOD

METHOD FB_init : BOOL
VAR_INPUT
	///if TRUE, the retain variables are initialized (warm start / cold start)
	bInitRetains: BOOL;
	///if TRUE, the instance afterwards gets moved into the copy code (online change)
	bInCopyCode: BOOL;
END_VAR
//------------------------------------------------------------------------------------------------------------------------
// enable cyclic call
me.bolActivate := TRUE;
// reset init flag
CIf.Info.bolInitDone := FALSE;

//------------------------------------------------------------------------------------------------------------------------
// to manually change in new FUB implementation!!!
// define valid commands for this controller
CIf.Job.aCmdList[0].intCmd := cCMD_PON;
CIf.Job.aCmdList[0].strName := 'Power On';
CIf.Job.aCmdList[0].bolAvailable := TRUE;

CIf.Job.aCmdList[1].intCmd := cCMD_OFF; // for test simulation single answer
CIf.Job.aCmdList[1].strName := 'Off';
CIf.Job.aCmdList[1].bolAvailable := TRUE;

CIf.Job.aCmdList[2].intCmd := cCMD_EOFF;
CIf.Job.aCmdList[2].strName := 'Emergency OFF';
CIf.Job.aCmdList[2].bolAvailable := TRUE;

// set name of class/typ
CIf.Info.strType := 'FB_CtrlBase'; 

// for tests
CIf.SwCfg.bolExist := TRUE;
CIf.SwCfg.bolSimulation := TRUE;

//------------------------------------------------------------------------------------------------------------------------
CIf.Info.strName := getStrInstanceName(strMyInstancePath); // get name of instance

CIf.Info.uinChildNbr := 0;
END_METHOD

METHOD PROTECTED getCmdState : STRING
VAR_INPUT
	intCmdState: INT;
	bolState: BOOL;
END_VAR
// get string cmd/state string information in runtime
IF (bolState=FALSE) THEN
	// cmd's
	CASE intCmdState OF
		cCMD_DONE: 
			getCmdState := 'cCMD_DONE';
		cCMD_INITIALIZED: 
			getCmdState := 'cCMD_INITIALIZED';
		cCMD_PON: 
			getCmdState := 'cCMD_PON';
		cCMD_EOFF: 
			getCmdState := 'cCMD_EOFF';
		cCMD_OFF: 
			getCmdState := 'cCMD_OFF';
		cCMD_INIT: 
			getCmdState := 'cCMD_INIT';
		cCMD_RUN: 
			getCmdState := 'cCMD_RUN';
		cCMD_STOP: 
			getCmdState := 'cCMD_STOP';
		cCMD_TSTOP: 
			getCmdState := 'cCMD_TSTOP';
	END_CASE;
ELSE

// cmd's
	CASE intCmdState OF
		cSTA_DONE: 
			getCmdState := 'cSTA_DONE';
		cSTA_INITIALIZED: 
			getCmdState := 'cSTA_INITIALIZED';
		cSTA_PONBusy: 
			getCmdState := 'cSTA_PONBusy';
		cSTA_PON: 
			getCmdState := 'cSTA_PON';
		cSTA_EOFFBusy: 
			getCmdState := 'cSTA_EOFFBusy';
		cSTA_EOFF: 
			getCmdState := 'cSTA_EOFF';
		cSTA_OFFBusy: 
			getCmdState := 'cSTA_OFFBusy';
		cSTA_OFF: 
			getCmdState := 'cSTA_OFF';
		cSTA_INITBusy: 
			getCmdState := 'cSTA_INITBusy';
		cSTA_INIT: 
			getCmdState := 'cSTA_INIT';
		cSTA_RUNBusy: 
			getCmdState := 'cSTA_RUNBusy';
		cSTA_RUN: 
			getCmdState := 'cSTA_RUN';
		cSTA_STOPBusy: 
			getCmdState := 'cSTA_STOPBusy';
		cSTA_STOP: 
			getCmdState := 'cSTA_STOP';
		cSTA_TSTOPBusy: 
			getCmdState := 'cSTA_TSTOPBusy';
		cSTA_TSTOP: 
			getCmdState := 'cSTA_TSTOP';
			
		cSTA_ERROR: 
			getCmdState := 'cSTA_ERROR';
		cSTA_ERRORQuit: 
			getCmdState := 'cSTA_ERRORQuit';
		cSTA_SINGLE_ANSWER: 
			getCmdState := 'cSTA_SINGLE_ANSWER';
	END_CASE;
END_IF
END_METHOD

METHOD PUBLIC iniAllCtrlArrays : BOOL
VAR_INPUT
	p_pCtrlFbBaseArray	: POINTER TO POINTER TO FB_CtrlBase;
	p_pCtrlCIfArray		: POINTER TO POINTER TO T_Ctrl_CIf;
	intCtrlID		: INT;
END_VAR
iniAllCtrlArrays := FALSE;

IF (TRUE) THEN//e_CtrlID <= E_CtrlId.E_CtrlIdMax) THEN
	p_pCtrlFbBaseArray[intCtrlID] 	:= THIS;
	THIS^.CIf.Info.intCtrlID := intCtrlID;
	p_pCtrlCIfArray[intCtrlID] := CtrlCIf;
	iniAllCtrlArrays := TRUE;
END_IF
END_METHOD

METHOD PROTECTED IoInBridge : BOOL
// digitale and analoge inputs read from hardware or forcing
IF (CIf.SwCfg.bolSimulation = FALSE) THEN
	//KVO??? alternative only without feedback getIn(ctrl.ifc.Job.bol_Force ,ADR(ctrl.In.bol_PosSwitchBasicDefTyp);
	//ctrl.In.bol_PosSwitchBasicDefTyp.intern := getIn(ctrl.ifc.Job.bol_Force ,ADR(ctrl.In.bol_PosSwitchBasicDefTyp);
ELSE
	//simulation of global IO
END_IF
END_METHOD

METHOD PROTECTED IoOutBridge : BOOL
// digitale and analoge inputs read from hardware or forcing
IF (CIf.SwCfg.bolSimulation = FALSE) THEN


//KVO??? alternative only without feedback getIn(ctrl.ifc.Job.bol_Force ,ADR(ctrl.In.bol_PosSwitchBasicDefTyp);
	// check interlocks to prevent damages
	//IF (SIf.Ilk.bolOverwrite=FALSE) THEN
		//IF (SIf.Ilk.bolOut=FALSE) THEN
			//ctrl.Out.bolOut.map := setOut(ctrl.ifc.Job.bol_Force ,ADR(ctrl.Out.bolOut);
		//ELSE
			// switch off???
			// error??
		//END_IF
	//end_if

	//THIS^.Out_bolOut := SIf.Out.bolOut.map;

END_IF
END_METHOD

METHOD PROTECTED SetAllChildAlmClass : BOOL
VAR_INPUT
	In_intSetAlmClass : INT;
END_VAR
VAR
	uinIdx: UINT;
END_VAR
IF (CIf.Info.uinChildNbr > 0) THEN
	FOR uinIdx := 0 TO CIf.Info.uinChildNbr - 1 DO
		CIf.Info.p_aCIf[uinIdx]^.Job.eParent_ActivAlmClass := In_intSetAlmClass;
	END_FOR
END_IF
END_METHOD

METHOD PROTECTED SetAllChildCmd
VAR_INPUT
	In_intSetAcmd : INT;
END_VAR
VAR
	uinIdx: UINT;
END_VAR
IF (CIf.Info.uinChildNbr > 0) THEN
	FOR uinIdx := 0 TO CIf.Info.uinChildNbr - 1 DO
		CIf.Info.p_aCIf[uinIdx]^.Job.intACmd := In_intSetAcmd;
	END_FOR
END_IF
END_METHOD

METHOD PROTECTED sta_EOFF : BOOL
VAR_INPUT
END_VAR
// state implemetation
//--------------------------------------------------------------------------------------
// Entry action
	IF (me.StateMachine.intState<>me.StateMachine.intStateLastCycle) THEN
		me.StateMachine.intStateLastCycle := me.StateMachine.intState;
		
	END_IF


//--------------------------------------------------------------------------------------
// Cyclic action
	IF (me.StateMachine.intState=me.StateMachine.intStateLastCycle) THEN
		
		;
		
		
		// State Change Condition
		IF (me.Alarm.eActivAlmClass<>E_AlmClass.EOFF) AND (me.intCmd<>cCMD_EOFF) AND (me.intCmd<>cCMD_DONE) THEN
			IF (FALSE) THEN
				;
			ELSIF (TRUE) THEN
				me.StateMachine.intStateNext := cSTA_OFF;
			END_IF
		END_IF
	END_IF




//--------------------------------------------------------------------------------------
// Exit action
	IF (me.StateMachine.intState<>me.StateMachine.intStateNext) THEN
		;
	END_IF
END_METHOD

METHOD PROTECTED sta_EOFFBusy : BOOL
VAR_INPUT
END_VAR
// state implemetation
//--------------------------------------------------------------------------------------
// Entry action
	IF (me.StateMachine.intState<>me.StateMachine.intStateLastCycle) THEN
		me.StateMachine.intStateLastCycle := me.StateMachine.intState;
		EOFF_EntryAction(); // used for special events in EOFF
		// Set commandos not only in entry action because of possible errors or manual/auto changes
		// PRE/AVME 06.01.2014
		//SetAllChildCmd(cCMD_EOFF); // set acmd off all childs 
	END_IF


//--------------------------------------------------------------------------------------
// Cyclic action
	IF (me.StateMachine.intState=me.StateMachine.intStateLastCycle) THEN
		
		SetAllChildCmd(cCMD_EOFF); // set acmd off all childs 
	
		// check if all childs have reached the state
		IF CheckAllChildState(cSTA_EOFF) THEN
			me.StateMachine.intStateNext := cSTA_EOFF;
		END_IF
	END_IF


//--------------------------------------------------------------------------------------
// Exit action
	IF (me.StateMachine.intState<>me.StateMachine.intStateNext) THEN
		;
	END_IF
END_METHOD

METHOD PROTECTED sta_ERROR : BOOL
// state implemetation
//--------------------------------------------------------------------------------------
// Entry action
	IF (me.StateMachine.intState<>me.StateMachine.intStateLastCycle) THEN
		me.StateMachine.intStateHistory := me.StateMachine.intStateLastCycle; // -> possibillity to go back to state before error
		me.StateMachine.intStateLastCycle := me.StateMachine.intState;
		
	END_IF


//--------------------------------------------------------------------------------------
// Cyclic action
	IF (me.StateMachine.intState=me.StateMachine.intStateLastCycle) THEN
		
		;
		
		
		// State Change Condition
		IF (CIf.Job.bolAlmReset = TRUE) THEN
			me.StateMachine.intStateNext := cSTA_ERRORQuit;
		END_IF
	END_IF




//--------------------------------------------------------------------------------------
// Exit action
	IF (me.StateMachine.intState<>me.StateMachine.intStateNext) THEN
		;
	END_IF
END_METHOD

METHOD PROTECTED sta_ERRORQuit : BOOL
// state implemetation
//--------------------------------------------------------------------------------------
// Entry action
	IF (me.StateMachine.intState<>me.StateMachine.intStateLastCycle) THEN
		me.StateMachine.intStateLastCycle := me.StateMachine.intState;
		
	END_IF


//--------------------------------------------------------------------------------------
// Cyclic action
	IF (me.StateMachine.intState=me.StateMachine.intStateLastCycle) THEN
		
		;
		// evtl. wait time if reset of device is necessary and then decide to go to states or ERROR state
		IF (CIf.Job.bolAlmReset = TRUE) THEN
			CIf.Job.eMe_ActivAlmClass := E_AlmClass.NONE; // reset feedback channel for parent
			CIf.Job.bolAlmReset := FALSE;
		END_IF
		
		// State Change Condition
		IF (CIf.Job.bolAlmReset = FALSE) OR (me.StateMachine.intStateHistory<=cSTA_PON) THEN
			me.StateMachine.intStateNext := cSTA_PONBusy;
		END_IF
	END_IF




//--------------------------------------------------------------------------------------
// Exit action
	IF (me.StateMachine.intState<>me.StateMachine.intStateNext) THEN
		;
	END_IF
END_METHOD

METHOD PROTECTED sta_OFF : BOOL
// state implemetation
//--------------------------------------------------------------------------------------
// Entry action
	IF (me.StateMachine.intState<>me.StateMachine.intStateLastCycle) THEN
		me.StateMachine.intStateLastCycle := me.StateMachine.intState;
		
	END_IF


//--------------------------------------------------------------------------------------
// Cyclic action
	IF (me.StateMachine.intState=me.StateMachine.intStateLastCycle) THEN
		
		;
		
		
		// State Change Condition
		IF ((me.Alarm.eActivAlmClass<>E_AlmClass.EOFF) AND (me.Alarm.eActivAlmClass<>E_AlmClass.OFF)) THEN
			IF (FALSE) THEN
				;
			ELSIF (TRUE) THEN
				;	//me.StateMachine.intStateNext := cSTA_PON;
			END_IF
		END_IF;
	END_IF




//--------------------------------------------------------------------------------------
// Exit action
	IF (me.StateMachine.intState<>me.StateMachine.intStateNext) THEN
		;
	END_IF
END_METHOD

METHOD PROTECTED sta_OFFBusy : BOOL
// state implemetation
//--------------------------------------------------------------------------------------
// Entry action
	IF (me.StateMachine.intState<>me.StateMachine.intStateLastCycle) THEN
		me.StateMachine.intStateLastCycle := me.StateMachine.intState;
		
		// Set commandos not only in entry action because of possible errors or manual/auto changes
		// PRE/AVME 06.01.2014
		//SetAllChildCmd(cCMD_OFF); // set acmd off all childs 
	END_IF


//--------------------------------------------------------------------------------------
// Cyclic action
	IF (me.StateMachine.intState=me.StateMachine.intStateLastCycle) THEN
		
		SetAllChildCmd(cCMD_OFF); // set acmd off all childs 
		
		// State Change Condition
		IF (FALSE) THEN
			;
		ELSIF (CheckAllChildState(cSTA_OFF)) THEN
			me.StateMachine.intStateNext := cSTA_OFF;
		END_IF
	END_IF




//--------------------------------------------------------------------------------------
// Exit action
	IF (me.StateMachine.intState<>me.StateMachine.intStateNext) THEN
		;
	END_IF
END_METHOD

METHOD PROTECTED sta_PON : BOOL
// state implemetation
//--------------------------------------------------------------------------------------
// Entry action
	IF (me.StateMachine.intState<>me.StateMachine.intStateLastCycle) THEN
		me.StateMachine.intStateLastCycle := me.StateMachine.intState;
		
	END_IF


//--------------------------------------------------------------------------------------
// Cyclic action
	IF (me.StateMachine.intState=me.StateMachine.intStateLastCycle) THEN
		
		;
		
		
		// State Change Condition
		IF (FALSE) THEN
			;
		ELSIF (me.intCmd<>cCMD_PON) AND (me.intCmd<>cCMD_DONE) THEN
			me.StateMachine.intStateNext := cSTA_EOFFBusy;
		END_IF
	END_IF




//--------------------------------------------------------------------------------------
// Exit action
	IF (me.StateMachine.intState<>me.StateMachine.intStateNext) THEN
		;
	END_IF
END_METHOD

METHOD PROTECTED sta_PONBusy : BOOL
// state implemetation
//--------------------------------------------------------------------------------------
// Entry action
	IF (me.StateMachine.intState<>me.StateMachine.intStateLastCycle) THEN
		me.StateMachine.intStateLastCycle := me.StateMachine.intState;
		
		SetAllChildCmd(cCMD_PON); // set acmd off all childs 
	END_IF


//--------------------------------------------------------------------------------------
// Cyclic action
	IF (me.StateMachine.intState=me.StateMachine.intStateLastCycle) THEN
		
		;
		
		
		// State Change Condition
		IF (FALSE) THEN
			;
		ELSIF CheckAllChildState(cSTA_PON) THEN
			me.StateMachine.intStateNext := cSTA_PON;
		END_IF
	END_IF




//--------------------------------------------------------------------------------------
// Exit action
	IF (me.StateMachine.intState<>me.StateMachine.intStateNext) THEN
		;
	END_IF
END_METHOD

METHOD PROTECTED sta_SINGLE_ANSWER : BOOL
// state implemetation of SINGLE_ANSWER
//--------------------------------------------------------------------------------------
// Entry action
	IF (me.StateMachine.intState<>me.StateMachine.intStateLastCycle) THEN
		me.StateMachine.intStateLastCycle := me.StateMachine.intState;
		
	END_IF


//--------------------------------------------------------------------------------------
// Cyclic action
	IF (me.StateMachine.intState=me.StateMachine.intStateLastCycle) THEN
		
		// Reset pending alarm class
		CIf.Job.eMe_ActivAlmClass := E_AlmClass.NONE;
	
		IF ((me.intCmd<>cCMD_INITIALIZED) AND (me.intCmd<>cCMD_DONE)) THEN
			IF (THIS^.CheckCmdValid()=TRUE) THEN
				IF (me.intCmd<>me.intCmdLast) THEN
					me.StateMachine.udiTimeInState_ms := 0;  // reset timer
				END_IF
				IF (me.StateMachine.udiTimeInState_ms >= me.StateMachine.udiStateSimSetTime_ms) THEN
					CIf.Job.intState := me.intCmd; // simulate final state
				ELSE
					CIf.Job.intState := me.intCmd-1; // simulate busy state
				END_IF
			END_IF
		END_IF
		
		// State Change Condition
		IF (FALSE) THEN
			;
		ELSIF (CIf.SwCfg.bolExist=TRUE) THEN
			me.StateMachine.intStateNext := cSTA_PONBusy;
		END_IF
	END_IF




//--------------------------------------------------------------------------------------
// Exit action
	IF (me.StateMachine.intState<>me.StateMachine.intStateNext) THEN
		;
	END_IF
END_METHOD

METHOD PROTECTED StateMachine : BOOL

// main statemachine of base controller
CASE me.StateMachine.intState OF
    cSTA_PONBusy: 
        THIS^.sta_PONBusy();
    cSTA_PON: 
        THIS^.sta_PON();
	cSTA_OFFBusy: 
        THIS^.sta_OFFBusy();
    cSTA_OFF: 
        THIS^.sta_OFF();
    cSTA_ERROR: 
        THIS^.sta_ERROR();
    cSTA_ERRORQuit: 
        THIS^.sta_ERRORQuit();
	cSTA_EOFFBusy:
		THIS^.sta_EOFFBusy();
	cSTA_EOFF:
		THIS^.sta_EOFF();
    cSTA_SINGLE_ANSWER: 
        THIS^.sta_SINGLE_ANSWER();
END_CASE;
END_METHOD

END_FUNCTION_BLOCK

// POUs/BaseCtrl/I_CtrlBase
INTERFACE I_CtrlBase

PROPERTY CtrlCIf : POINTER TO T_Ctrl_CIf
GET
END_GET
END_PROPERTY

PROPERTY CtrlFB : POINTER TO FB_CtrlBASE
GET
END_GET
END_PROPERTY

END_INTERFACE

// POUs/Utility/getStrInstanceName
FUNCTION getStrInstanceName : T_MaxString
VAR_INPUT
	///'C:\TwinCAT\Plc\Project01\Data.txt';
	strPathName: T_MaxString;
END_VAR
VAR
	strDrive: STRING(3);
	strDir: T_MaxString;
	strFileName: T_MaxString;
	strExt: T_MaxString;
	bolSuccess: BOOL;
END_VAR


bolSuccess := F_SplitPathName( sPathName := strPathName,
                                sDrive := strDrive,
                                sDir := strDir,
                                sFileName := strFileName,
                                sExt := strExt );
								
								getStrInstanceName := MID (strExt,TC2_STANDARD.LEN(strExt),2);

END_FUNCTION

// POUs/Utility/DLL (Double Linked List)/FB_DLL
FUNCTION_BLOCK FB_DLL
VAR
	bDoDataWipe: BOOL := FALSE;
	pFirstElement: POINTER TO T_Element;
	pLastElement: POINTER TO T_Element;
	uiNumberOfElements: UINT;
END_VAR

METHOD addElement : POINTER TO T_Element
VAR_INPUT
	In_pData: POINTER TO BYTE;
	In_uliKey: ULINT;
END_VAR
VAR
	pCurrentElement: POINTER TO T_Element;
END_VAR
addElement := TC3_MEMMAN.NULL;

IF (pFirstElement = TC3_MEMMAN.NULL) THEN
	pCurrentElement := __NEW(T_Element);
	pFirstElement := pCurrentElement;
	pLastElement := pCurrentElement;
	pCurrentElement^.pPrevElement := TC3_MEMMAN.NULL;
	pCurrentElement^.pNextElement := TC3_MEMMAN.NULL;
	pCurrentElement^.pData := In_pData;
	pCurrentElement^.uliKey := In_uliKey;
	addElement := pCurrentElement;
ELSE
	pCurrentElement := __NEW(T_Element);
	pCurrentElement^.pPrevElement := pLastElement;
	pCurrentElement^.pNextElement := TC3_MEMMAN.NULL;
	pCurrentElement^.pData := In_pData;
	pCurrentElement^.uliKey := In_uliKey;
	pLastElement^.pNextElement := pCurrentElement;
	pLastElement := pCurrentElement;
	addElement := pCurrentElement;
END_IF

uiNumberOfElements := uiNumberOfElements + 1;
END_METHOD

METHOD deleteAll : POINTER TO T_Element
WHILE (pFirstElement <> TC3_MEMMAN.NULL) DO
	__DELETE(pFirstElement^.pData);
	deleteElement(pFirstElement);
END_WHILE
END_METHOD

METHOD deleteElement : POINTER TO BYTE
VAR_INPUT
	In_pDeleteElement: POINTER TO T_Element;
END_VAR
deleteElement := In_pDeleteElement^.pData;

IF bDoDataWipe THEN
	IF (In_pDeleteElement^.pData <> TC3_MEMMAN.NULL) THEN
		__DELETE(In_pDeleteElement^.pData);
	END_IF
	deleteElement := TC3_MEMMAN.NULL;
END_IF

IF (In_pDeleteElement = pFirstElement AND In_pDeleteElement = pLastElement) THEN
	pFirstElement := TC3_MEMMAN.NULL;
	pLastElement := TC3_MEMMAN.NULL;
ELSIF (In_pDeleteElement = pFirstElement) THEN
	pFirstElement := In_pDeleteElement^.pNextElement;
	In_pDeleteElement^.pNextElement^.pPrevElement := TC3_MEMMAN.NULL;
ELSIF (In_pDeleteElement = pLastElement) THEN
	pLastElement := In_pDeleteElement^.pPrevElement;
	In_pDeleteElement^.pPrevElement^.pNextElement := TC3_MEMMAN.NULL;
ELSE
	In_pDeleteElement^.pPrevElement^.pNextElement := In_pDeleteElement^.pNextElement;
	In_pDeleteElement^.pNextElement^.pPrevElement := In_pDeleteElement^.pPrevElement;
END_IF

__DELETE(In_pDeleteElement);

uiNumberOfElements := uiNumberOfElements - 1;
END_METHOD

METHOD FB_init : BOOL
VAR_INPUT
	/// if TRUE, the retain variables are initialized (warm start / cold start)
	bInitRetains: BOOL;
	/// if TRUE, the instance afterwards gets moved into the copy code (online change)
	bInCopyCode: BOOL;
	/// if TRUE, the stored data object are automatically deleted
	In_bDoDataWipe: BOOL;
END_VAR
pFirstElement := TC3_MEMMAN.NULL;
pLastElement := TC3_MEMMAN.NULL;
uiNumberOfElements := 0;

bDoDataWipe := In_bDoDataWipe;
END_METHOD

METHOD firstElement : POINTER TO T_Element
firstElement := pFirstElement;
END_METHOD

METHOD numberOfElements : UINT
numberOfElements := uiNumberOfElements;
END_METHOD

METHOD searchElement : POINTER TO T_Element
VAR_INPUT
	In_uliKey: ULINT;
END_VAR
VAR
	pCurrentElement: POINTER TO T_Element;
END_VAR
searchElement := TC3_MEMMAN.NULL;
pCurrentElement := pFirstElement;

WHILE (pCurrentElement <> TC3_MEMMAN.NULL) DO
	IF (pCurrentElement^.uliKey = In_uliKey) THEN
		searchElement := pCurrentElement;
		EXIT;
	END_IF
	pCurrentElement := pCurrentElement^.pNextElement;
END_WHILE
END_METHOD

END_FUNCTION_BLOCK

// POUs/Utility/getInBol
FUNCTION getInBol : BOOL
VAR_INPUT
	bol_GlobalEnableForce: BOOL;
	p_Input: POINTER TO T_Ctrl_IoBool;
END_VAR

p_Input^.state := p_Input^.map;

IF (p_Input^.EnForce AND bol_GlobalEnableForce) THEN
	p_Input^.intern := p_Input^.force;
ELSE
	p_Input^.intern := p_Input^.map;
END_IF;

getInBol := p_Input^.intern;

END_FUNCTION

// POUs/Utility/getInBolDebounced
FUNCTION getInBolDebounced : BOOL
VAR_INPUT
	bol_GlobalEnableForce: BOOL;
	udiSample_ms: UDINT;		// Sample time from me.FUBInfo.udiSample_ms
	udiDebounceTime_ms: UDINT;	// Wait time for debouncing in ms
	p_Input: POINTER TO T_Ctrl_IoBoolDebounced;
END_VAR

// The input is accepted only after the debounce time (udiDebounceTime_ms)
// If the signal changes during this time, the timer will be restarted

IF (p_Input^.EnForce AND bol_GlobalEnableForce) THEN	// Forced signal, no debouncing neccessary
	p_Input^.intern := p_Input^.force;
ELSE													// Debounce signal
	IF p_Input^.state <> p_Input^.map THEN
		p_Input^.udinDebouncedTimeCounter_ms := 0;
	END_IF
	IF p_Input^.udinDebouncedTimeCounter_ms < udiDebounceTime_ms THEN
		p_Input^.udinDebouncedTimeCounter_ms := p_Input^.udinDebouncedTimeCounter_ms + udiSample_ms;
	ELSE
		p_Input^.intern := p_Input^.map;		
	END_IF
END_IF;

p_Input^.state := p_Input^.map;

getInBolDebounced := p_Input^.intern;

END_FUNCTION

// POUs/Utility/getInInt
FUNCTION getInInt : INT
VAR_INPUT
	bol_GlobalEnableForce: BOOL;
	p_Input: POINTER TO T_Ctrl_IoInt;
END_VAR

p_Input^.state := p_Input^.map;

IF (p_Input^.EnForce AND bol_GlobalEnableForce) THEN
	p_Input^.intern := p_Input^.force;
ELSE
	p_Input^.intern := p_Input^.map;
END_IF;

getInInt := p_Input^.intern;

END_FUNCTION

// POUs/Utility/getInUint
FUNCTION getInUint : UINT
VAR_INPUT
	bol_GlobalEnableForce		: BOOL;
	p_Input						: POINTER TO T_Ctrl_IoUint;
END_VAR
VAR
END_VAR

p_Input^.state := p_Input^.map;

IF (p_Input^.EnForce AND bol_GlobalEnableForce) THEN
	p_Input^.intern := p_Input^.force;
ELSE
	p_Input^.intern := p_Input^.map;
END_IF;

getInUint := p_Input^.intern;

END_FUNCTION

// POUs/Utility/getInUsint
FUNCTION getInUsint : USINT
VAR_INPUT
	bol_GlobalEnableForce		: BOOL;
	p_Input						: POINTER TO T_Ctrl_IoUsint;
END_VAR
VAR
END_VAR

p_Input^.state := p_Input^.map;

IF (p_Input^.EnForce AND bol_GlobalEnableForce) THEN
	p_Input^.intern := p_Input^.force;
ELSE
	p_Input^.intern := p_Input^.map;
END_IF;

getInUsint := p_Input^.intern;

END_FUNCTION

// POUs/Utility/ScaleINT
FUNCTION ScaleINT : INT //Output signal.
VAR_INPUT
	x: INT; 	// Input signal. Allowed values: -32768..+32767.
	x1 : INT;	// Abscissa for the 1st coordinate. Allowed values: -32768..+32767
	x2 : INT;	// Abscissa for the 2nd coordinate. Allowed values: -32768..+32767.
	y1 : INT;	// Ordinate for the 1st coordinate. First limit of the value range. Allowed values: –32768..+32767.
	y2: INT;	// Ordinate for the 2nd coordinate. Second limit of the value range. Allowed values: -32768..+32767.
END_VAR
VAR
END_VAR


(*	IF x1 = x2, THEN 0 is output *)

// Scale value 
IF (x1=x2) THEN // -> zero division!
	ScaleINT := 0;
ELSE
	ScaleINT := (((x - x1) * (y2-y1))/(x2-x1)) + y1;
END_IF

END_FUNCTION

// POUs/Utility/setAllCtrlAlarmFB
FUNCTION setAllCtrlAlarmFB : BOOL
VAR_INPUT
	pCtrlInst			: POINTER TO POINTER TO FB_CtrlBase;
	pAlarmCtrl			: POINTER TO FB_Alm_Man;
	uinCtrlInstLength	: UINT;
END_VAR
VAR
	uinIdx	: UINT;
END_VAR

FOR uinIdx := 0 TO uinCtrlInstLength DO
	IF pCtrlInst[uinIdx] <> 0 THEN
		pCtrlInst[uinIdx]^.AlarmCtrl := pAlarmCtrl;
	END_IF
END_FOR

END_FUNCTION

// POUs/Utility/setOutBol
FUNCTION setOutBol : BOOL
VAR_INPUT
	bol_GlobalEnableForce: BOOL;
	p_Output: POINTER TO T_Ctrl_IoBool;
END_VAR

// Copy real values
p_Output^.state := p_Output^.intern;

IF (p_Output^.EnForce AND bol_GlobalEnableForce) THEN
	p_Output^.map := p_Output^.force;
ELSE
	p_Output^.map := p_Output^.intern;
END_IF;

setOutBol := p_Output^.map;

END_FUNCTION

// POUs/Utility/setOutInt
FUNCTION setOutInt : INT
VAR_INPUT
	bol_GlobalEnableForce: BOOL;
	p_Output: POINTER TO T_Ctrl_IoInt;
END_VAR

// Copy real values
p_Output^.state := p_Output^.intern;

IF (p_Output^.EnForce AND bol_GlobalEnableForce) THEN
	p_Output^.map := p_Output^.force;
ELSE
	p_Output^.map := p_Output^.intern;
END_IF;

setOutInt := p_Output^.map;

END_FUNCTION

// POUs/Utility/setOutUint
FUNCTION setOutUint : UINT
VAR_INPUT
	bol_GlobalEnableForce	: BOOL;
	p_Output				: POINTER TO T_Ctrl_IoUint;
END_VAR
VAR
END_VAR

// Copy real values
p_Output^.state := p_Output^.intern;

IF (p_Output^.EnForce AND bol_GlobalEnableForce) THEN
	p_Output^.map := p_Output^.force;
ELSE
	p_Output^.map := p_Output^.intern;
END_IF;

setOutUint := p_Output^.map;

END_FUNCTION

// POUs/Utility/setOutUsint
FUNCTION setOutUsint : USINT
VAR_INPUT
	bol_GlobalEnableForce	: BOOL;
	p_Output				: POINTER TO T_Ctrl_IoUsint;
END_VAR
VAR
END_VAR

// Copy real values
p_Output^.state := p_Output^.intern;

IF (p_Output^.EnForce AND bol_GlobalEnableForce) THEN
	p_Output^.map := p_Output^.force;
ELSE
	p_Output^.map := p_Output^.intern;
END_IF;

setOutUsint := p_Output^.map;

END_FUNCTION
